PROGRAM MAIN
VAR
END_VAR

P_Unit_Tests();

END_PROGRAM

(* stored: Version 1.1.0.1, ProductVersion 3.1.4022.7
   POU MAIN: Id {bd0d55d2-1d88-47bc-a7ac-f3fc8e9c2c35}, SpecialFunc None *)
